FUNCTION_BLOCK FB_STI_Conveyor_V2 IMPLEMENTS ITF_SubsystemTransport
(**************************************************************************************
 * 	Application		:	BoxControl Framework
 *	Revision		:	$Revision: 355211 $
 *	Revision date	:	$Date: 2015-09-22 11:14:21 +0200 (Tue, 22 Sep 2015) $
 *	Last changed by	:	$Author: d7mangc $
 *	URL				:	$URL: http://almscdc.swisslog.com/repo/SWPD/Development/BoxControlFramework/20_Release/trunk/01_Software/BoxControlFramework/BoxControlFramework/JumpStart/11_Library/10_Application/11_Communication/12_MFCS/11_SIS/10_Base/FB_SIS_BaseDriver.TcPOU $
 *
 *	Purpose			:	Subsystem transport interface: Conveyor
 *
 * ------------------------------------------------------------------------------------
 *	Copyright Swisslog [IP AG], Switzerland. All rights reserved.
 * 
 * ------------------------------------------------------------------------------------
 *	
 * 	Revision History: 
 *
 * VERSION DATE         INITIALS     DESCRIPTION
 * 0.0     DD.MM.YYYY   (name)       (explain customized modifications)
 *
 **************************************************************************************)
VAR_INPUT
	Config					: ST_CFG_STI_Conveyor; // Config
END_VAR
VAR_OUTPUT
	Outputs					: ST_InOutputsSTI_Conveyor; // Outputs
END_VAR
VAR
	Init					: BOOL; // Initialize
	fbDebugMsg				: FB_DebugMsg; // Debug instance
	DebugMsg				: T_MAXSTRING; // Debug msg
	fbTCP_Driver			: FB_TCP_Driver;
	ErrorData				: ST_ErrorDataSet; // Error data
	DestinationPosition		: ST_PositionIdent; 
	Position				: ST_PositionIdent; 
	ExternalTU_DataIndex	: DINT; 
	TU_DataIndex			: DINT;
	TU_DataIndexAssignment	: DINT;
	LastHandoverTU_DataIndex: DINT;
	TransportControlData	: ST_TransportControlData; 
	eHandOverState			: E_HandoverState; // Handover state machine
	eLastHandOverState		: E_HandoverState; // Handover state machine
	eTakeOverState			: E_TakeoverState; // Takeover state machine
	eLastTakeOverState		: E_TakeoverState; // Takeover state machine
	Inputs					: ST_InOutputsSTI_Conveyor; // Input structure
	AdjTransportData		: ST_TransportData; // Transport data of adjacent function
	RecvByte				: ARRAY[1..38] OF BYTE; // Receive as bytes (alignment)
	SendByte				: ARRAY[1..38] OF BYTE; // Send as bytes (alignment)
	RecvData				: ST_STI_ConveyorData; // Incoming conveyor data
	SendData				: ST_STI_ConveyorData; // Outgoing conveyor data
	LastSendData			: ST_STI_ConveyorData; // Last outgoing conveyor data
	ReceivedDataLen			: UDINT; // Received length
	RecvCounter				: USINT; // Counts received messages
	SendCounter				: USINT; // Counts sent messages
	fbWatchdogTimer			: TON; // Monitors watchdog signal
	fbReinitConnection		: TON; // Timer connection retry
	fbResend				: TON; // Timer for resending last message
	fbHeartBeatTimer		: TON; // Timer for generating heart beat of watchdog
	TransportData			: ST_TransportData; // Transport data
	DataError				: BOOL; // Error on data allocation action
	FlagWatchdog			: BOOL; // Flag, to save last watchdog state
	tHeartBeat				: TIME; // Time for generating watchdog heart beat
	TU_ID_Present			: BOOL; // TU ID present
	AssignmentID_Present	: BOOL; // Assignment ID present
	NewIndexCreated			: BOOL;
	TTC						: ST_ITC_TTC; // TTC
END_VAR
VAR PERSISTENT
	Settings				: ST_CFG_STI_Conveyor;
END_VAR

(**************************************************************************************************************
   Body never called!
***************************************************************************************************************)
;

ACTION A_AllocateDataIndex:
(**************************************************************************************
 * 	NAME		A_AllocateDataIndex
 * 	FUNCTION	Allocate a data index
 **************************************************************************************)

 (**************************************************************************************
   Delete old
***************************************************************************************)
 // If an old index is still available
 IF ExternalTU_DataIndex <> 0 THEN
	// Check if a position contains this index
	Position := F_SearchPositionOfTU_Index(
					TU_DataIndex := ExternalTU_DataIndex,
					eStartFunctionNumber := E_FunctionNumber.F_BEGIN_FUNCTION);
					
	// If index was found on a position
	IF Position.eFunctionNumber > E_FunctionNumber.F_BEGIN_FUNCTION THEN
		// debug message: '11-001-0000-00-0,  used TU_DataIndex deleted, position = 99-999-9999-99-9,  TU_DataIndex = 5,  TuID = 000012345,  AssignmentID = 999999999'
		DebugMsg := '';
		DebugMsg := CONCAT(DebugMsg, F_AddDividerToSisString(SubsystemRegistry.SubsystemName));
		DebugMsg := CONCAT(DebugMsg, ',  used TU_DataIndex deleted');
		DebugMsg := CONCAT(DebugMsg, DebugTextBlocks.POSITION);
		DebugMsg := CONCAT(DebugMsg, Position.PositionName);
		DebugMsg := CONCAT(DebugMsg, F_CreateTU_DataString(TU_DataIndex:= ExternalTU_DataIndex));
		fbDebugMsg.M_SendWarningMsg(mMessage := DebugMsg);
		
		// Clear only index
		ExternalTU_DataIndex := 0;
	ELSE
		// debug message: '11-000-0000-00-0,  unused TU_DataIndex deleted, external = 99-999-9999-99-9,  TU_DataIndex = 5,  TuID = 000012345,  AssignmentID = 999999999'
		DebugMsg := '';
		DebugMsg := CONCAT(DebugMsg, F_AddDividerToSisString(SubsystemRegistry.SubsystemName));
		DebugMsg := CONCAT(DebugMsg, ',  unused TU_DataIndex deleted');
		DebugMsg := CONCAT(DebugMsg, DebugTextBlocks.POSITION);
		DebugMsg := CONCAT(DebugMsg, TO_STRING(Settings.eExternalFunctionNumber));  // ###todo: how to retrieve sis number string for external?
		DebugMsg := CONCAT(DebugMsg, F_CreateTU_DataString(TU_DataIndex:= ExternalTU_DataIndex));
		fbDebugMsg.M_SendInfoMsg(DebugMsg);
		// Clear data set
		F_DeleteTU_Data(
			TU_DataIndex 	:= ExternalTU_DataIndex,
			NoTTC 			:= TRUE);
			
		// Clear index
		ExternalTU_DataIndex := 0;
	END_IF
 END_IF
 
 (**************************************************************************************
   Allocate new index
***************************************************************************************)
TU_ID_Present := Inputs.TU_ID <> '000000000000000000' AND
				 Inputs.TU_ID <> '                  ' AND
			 	 Inputs.TU_ID <> '';

AssignmentID_Present := Inputs.AssignmentID > 0;

// If giving conveyor provides a TU ID or an assignment ID
IF TU_ID_Present OR
   AssignmentID_Present THEN
   
   // Reset
   DataError := FALSE;
   
	// Search if index based on TU-ID is already available 
	TU_DataIndex := F_SearchTU_ByHashCode(TU_ID := Inputs.TU_ID);
	// Search if index based on Assignment is already available
	TU_DataIndexAssignment := F_SearchAssignmentId(Inputs.AssignmentID);

	// When both an index for the TU-ID AND the Assignment ID is available in the system 
	IF TU_DataIndex > 0 AND TU_DataIndexAssignment > 0 THEN
		// Check if they are equal, otherwise data set is ignored
		// This would lead to a data mismatch.
		IF TU_DataIndex <> TU_DataIndexAssignment THEN
		   DataError := TRUE;
		   
		   	// Debug - wrong index found
			DebugMsg := CONCAT('External interface: AssignmentID and TU-ID have not the same index. TU-ID index:', DINT_TO_STRING(TU_DataIndex));
			DebugMsg := CONCAT(DebugMsg, ', AssignmentID index: ');
			DebugMsg := CONCAT(DebugMsg, DINT_TO_STRING(TU_DataIndexAssignment));
			fbDebugMsg.M_SendWarningMsg(mMessage := DebugMsg);
		
		// Clear TU slot before taking over TU data from the Interface
		ELSIF Settings.DeleteTU_Data THEN
			MEMSET(ADR(TU_DataTable[TU_DataIndex]), 0, SIZEOF(TU_DataTable[TU_DataIndex]));	
		END_IF 
		
	// When index for TU-ID OR  Assignment ID is available in the system
	ELSIF TU_DataIndex > 0  OR TU_DataIndexAssignment > 0 THEN
		
		IF Settings.DeleteTU_Data THEN
			// Clear TU slot before taking over TU data from the Interface
			MEMSET(ADR(TU_DataTable[TU_DataIndex]), 0, SIZEOF(TU_DataTable[TU_DataIndex]));	
		END_IF 
		
	// When index for Assignment ID is available in the system
	ELSIF TU_DataIndexAssignment > 0 THEN
		IF Settings.DeleteTU_Data THEN
			// Clear TU slot before taking over TU data from the Interface
			MEMSET(ADR(TU_DataTable[TU_DataIndexAssignment]), 0, SIZEOF(TU_DataTable[TU_DataIndexAssignment]));	
		END_IF 	
		TU_DataIndex := TU_DataIndexAssignment; 	
		
	ELSE
		// Allocate new one
	   TU_DataIndex := F_InsertTU_Data(
							eFunctionNumber := Settings.AdjFunctionNumber.eFunctionNumber,
							ZoneNumber := Settings.AdjFunctionNumber.ZoneNumber);
		
		NewIndexCreated := TU_DataIndex > 0;		
		
		// If creation was not succesfull
		IF NOT NewIndexCreated THEN
			DataError := TRUE;
		   
		   	// Debug - Image creation failed
			DebugMsg := 'External interface: AllocateDataIndex was not able to create free index';
			fbDebugMsg.M_SendWarningMsg(mMessage := DebugMsg);
			
			// Error no free TU Index
			IF ErrorData.ErrorType = E_ErrorType.NO_ERROR_PENDING THEN
				// Set communication error
				F_SetError(
					ErrorMsg	:= E_ErrorConv.NO_FREE_TU_DATA_SET,
					ErrorType 	:= E_ErrorType.ERROR,
					ErrorParam 	:= '',
					ErrorData	:= ErrorData);
			END_IF
		END_IF
	END_IF
   
	// When no error occured 
	IF NOT DataError AND 
		TU_DataIndex > 0 THEN
		
		//  when new Tu data index was created or exisitng should be overwritten
		IF	Settings.OverwriteTU_Data OR NewIndexCreated THEN
			//Takeover data from interface
			
			// Set data present
			TU_DataTable[TU_DataIndex].DataSet.DataPresent := TRUE;
			
			// Update data
			IF TU_ID_Present THEN
				TU_DataTable[TU_DataIndex].TU_ID.ASCII := Inputs.TU_ID;
				TU_DataTable[TU_DataIndex].TU_ID.HashCode := F_CreateHashCode(Inputs.TU_ID);
			END_IF
			
			IF AssignmentID_Present THEN
				TU_DataTable[TU_DataIndex].AssignmentID := Inputs.AssignmentID;
			END_IF
	
			IF Inputs.Destination <> '' THEN
				// Search function number of corresponding string
				DestinationPosition := F_SearchFunctionPosition(Position := Inputs.Destination);
			
				// Destination was found 
				IF DestinationPosition.eFunctionNumber <> 0 THEN
					TU_DataTable[TU_DataIndex].Destination[1].eFunctionNumber 	:= DestinationPosition.eFunctionNumber;
					TU_DataTable[TU_DataIndex].Destination[1].ZoneNumber 		:= DestinationPosition.ZoneNumber;
					TU_DataTable[TU_DataIndex].Destination[1].PositionName 		:= DestinationPosition.PositionName;
					TU_DataTable[TU_DataIndex].DataSet.JobPresent := TRUE;
					TU_DataTable[TU_DataIndex].DataSet.NumberOfDest := 1;
				ELSE
					// Debug - Destination not found
					DebugMsg := CONCAT('External interface: Destination not found(', Inputs.Destination);
					DebugMsg := CONCAT(DebugMsg, ')');
					
					fbDebugMsg.M_SendWarningMsg(mMessage := DebugMsg);
				END_IF
			END_IF			
		END_IF
		// Set to external TU Data Index
		ExternalTU_DataIndex := TU_DataIndex;
	END_IF
END_IF
END_ACTION

ACTION A_HandOverStates:
(**************************************************************************************
 * 	NAME		A_HandOverInterface
 * 	FUNCTION	Handover interface
 **************************************************************************************)

(**************************************************************************************
	Update outputs for external conveyor position
**************************************************************************************)
Outputs.ReadyToTakeOver := AdjTransportData.rTransportControlData.eTakeOverState = E_TakeOverState.READY OR
						   AdjTransportData.rTransportControlData.eTakeOverState = E_TakeOverState.INTERRUPTED;

Outputs.TakeoverStarted := AdjTransportData.rTransportControlData.eTakeOverState = E_TakeOverState.ACTIVE OR
						   AdjTransportData.rTransportControlData.eTakeOverState = E_TakeOverState.INTERRUPTED OR
						   AdjTransportData.rTransportControlData.eTakeOverState = E_TakeOverState.STOP OR
						   AdjTransportData.rTransportControlData.eTakeOverState = E_TakeOverState.COMPLETE;

Outputs.TakeoverActive := AdjTransportData.rTransportControlData.eTakeOverState = E_TakeOverState.ACTIVE;
						  
Outputs.TakeoverComplete := AdjTransportData.rTransportControlData.eTakeOverState = E_TakeOverState.COMPLETE;

Outputs.TransportActive := AdjTransportData.rTransportControlData.TransportActive;
Outputs.FastSpeedActive := AdjTransportData.rTransportControlData.FastSpeedActive;

(**************************************************************************************
	Simulates hand over state for external conveyor position
 **************************************************************************************)
CASE eHandOverState OF
	
	(**********************************************************************************
	   BEGIN
	***********************************************************************************)
	E_HandOverState.UNDEFINED:
	
		// Change state to "IDLE"
		eLastHandOverState := eHandOverState;
		eHandOverState := E_HandOverState.IDLE;
	
	(**********************************************************************************
	   IDLE
	***********************************************************************************)
	E_HandOverState.IDLE:

		// If external interface is ready to hand over
		IF Inputs.ReadyToHandOver THEN
			// Allocate data index
			A_AllocateDataIndex();
		
			// Change state to "IDLE"
			eLastHandOverState := eHandOverState;
			eHandOverState := E_HandOverState.READY;
		END_IF
	
	(**********************************************************************************
	   READY
	***********************************************************************************)
	E_HandOverState.READY:
	
		IF Inputs.HandoverActive THEN
			// Change state to "ACTIVE"
			eLastHandOverState := eHandOverState;
			eHandOverState := E_HandOverState.ACTIVE;
	
		// If external interface is not ready for hand over
		ELSIF NOT Inputs.ReadyToHandOver THEN
			// Go back to state to "IDLE"
			eLastHandOverState := eHandOverState;
			eHandOverState := E_HandOverState.IDLE;
		END_IF
		
	(**********************************************************************************
	   ACTIVE
	***********************************************************************************)
	E_HandOverState.ACTIVE:
	
		// Wait until completed
		IF Inputs.HandoverComplete THEN
			// Change state to "COMPLETE"
			eLastHandOverState := eHandOverState;
			eHandOverState := E_HandOverState.COMPLETE;
		
		// If handover is not active anymore
		ELSIF NOT Inputs.HandoverActive THEN
			// Ready already set -> Takeover conveyor stopped handover
			IF Inputs.ReadyToHandover THEN
				// Change state to "Interrupted"
				eLastHandOverState := eHandOverState;
				eHandOverState := E_HandOverState.INTERRUPTED;
				
			// Otherwise the external conveyor has stopped the handover
			ELSE
				// If the handover task is the same - was an error during transport -> Stop
				IF Inputs.HandoverStarted THEN
					// Change state to "Stop"
					eLastHandOverState := eHandOverState;
					eHandOverState := E_HandOverState.STOP;
					
				// Otherwise transport was aborted completely
				ELSE
					// Change state to "Idle"
					eLastHandOverState := eHandOverState;
					eHandOverState := E_HandOverState.IDLE;
				END_IF
			END_IF
		END_IF
	
	(**********************************************************************************
	   STOP
	***********************************************************************************)
	E_HandOverState.STOP:
			
		// Wait until transfer goes on 
		IF Inputs.HandoverActive THEN
			// Change state to "ACTIVE"
			eLastHandOverState := eHandOverState;
			eHandOverState := E_HandOverState.ACTIVE;

		// If the handover is completed 
		ELSIF Inputs.HandoverComplete THEN
			// Change state to "ACTIVE"
			eLastHandOverState := eHandOverState;
			eHandOverState := E_HandOverState.COMPLETE;	
		
		// If the ongoing transport task was aborted
		ELSIF NOT Inputs.HandoverStarted THEN
			// Change state to "Idle"
			eLastHandOverState := eHandOverState;
			eHandOverState := E_HandOverState.IDLE;
		END_IF
	
	(**********************************************************************************
	   INTERRUPTED
	***********************************************************************************)
	E_HandOverState.INTERRUPTED:
	
		// Wait until hadover is active
		IF Inputs.HandoverActive THEN
			// Change state to "ACTIVE"
			eLastHandOverState := eHandOverState;
			eHandOverState := E_HandOverState.ACTIVE;
			
		// If the handover is completed 
		ELSIF Inputs.HandoverComplete THEN
			// Change state to "ACTIVE"
			eLastHandOverState := eHandOverState;
			eHandOverState := E_HandOverState.COMPLETE;				
			
		// If the ongoing transport task was aborted
		ELSIF NOT Inputs.HandoverStarted THEN
			// Change state to "Idle"
			eLastHandOverState := eHandOverState;
			eHandOverState := E_HandOverState.IDLE;
		END_IF
		
	(**********************************************************************************
	   COMPLETE
	***********************************************************************************)
	E_HandOverState.COMPLETE:
	
		// Wait until transfer complete signal is resetted
		IF NOT Inputs.HandoverComplete OR
           NOT Inputs.HandoverStarted THEN
			// Change state to "IDLE"
			eLastHandOverState := eHandOverState;
			eHandOverState := E_HandOverState.IDLE;
		END_IF 
		
ELSE
	// Programming error
	DebugMsg := CONCAT(	'Programming error - Invalid state of external interface (Handover): ', 
					   	INT_TO_STRING(eHandOverState));
	DebugMsg := CONCAT(	DebugMsg, ' External connection : ');
	DebugMsg := CONCAT(	DebugMsg, INT_TO_STRING(Settings.eExternalFunctionNumber));
	fbDebugMsg.M_SendErrorMsg(DebugMsg);
END_CASE
END_ACTION

ACTION A_InputMapping:
(**************************************************************************************
 * 	NAME		A_InputMapping
 * 	FUNCTION	Map input variables
 **************************************************************************************)

(**************************************************************************************
   Map interface inputs
***************************************************************************************)
 
// If interface is configured as inbound
IF Settings.Inbound THEN
	Inputs.HandoverActive := RecvData.HandoverActive;
	Inputs.HandoverComplete := RecvData.HandoverComplete;
	Inputs.ReadyToHandover := RecvData.ReadyToHandover;	
	Inputs.HandoverStarted := RecvData.HandoverStarted;
	Inputs.TakeoverActive := FALSE;
	Inputs.TakeoverComplete := FALSE;
	Inputs.ReadyToTakeover := FALSE;
	Inputs.TakeoverStarted := FALSE;
	
// Otherwise, outbound
ELSE
	Inputs.TakeoverActive := RecvData.TakeoverActive;
	Inputs.TakeoverComplete := RecvData.TakeoverComplete;
	Inputs.ReadyToTakeover := RecvData.ReadyToTakeover;
	Inputs.TakeoverStarted := RecvData.TakeoverStarted;
	Inputs.HandoverActive := FALSE;
	Inputs.HandoverComplete := FALSE;
	Inputs.ReadyToHandover := FALSE;	
	Inputs.HandoverStarted := FALSE;
END_IF

// General data
Inputs.TU_ID := RecvData.TU_Data.TU_ID;
Inputs.AssignmentID := RecvData.TU_Data.AssignmentID;
Inputs.Destination := RecvData.TU_Data.Destination;

IF Settings.OnlyFastSpeed THEN
	Inputs.FastSpeedActive := TRUE;
ELSE
	Inputs.FastSpeedActive := RecvData.FastSpeedActive;
END_IF

Inputs.TransportActive := RecvData.TransportActive;

(**************************************************************************************
   Get external data
***************************************************************************************)
// Get transport data of adjacent function
AdjTransportData := F_GetAdjacentTransportData(
						eFunctionNumber 		:= Settings.AdjFunctionNumber.eFunctionNumber,
						eSourceFunctionNumber 	:= Settings.eExternalFunctionNumber);
END_ACTION

ACTION A_MonitorCommunication:
(**************************************************************************************
 * 	NAME		A_MonitorCommunication
 * 	FUNCTION	Monitors TCP Communication
 **************************************************************************************)

(**************************************************************************************
   Watchdog
***************************************************************************************) 
fbWatchdogTimer(IN := TRUE, PT := Settings.tWatchdog);
 
// If connection is server
IF Settings.TCP_Driver.Server THEN
	// Watchdog signals
	IF RecvData.WatchdogToggle = SendData.WatchdogToggle THEN
		// Reset timer
		fbWatchdogTimer(IN := FALSE);
		fbHeartBeatTimer(IN := TRUE, PT := tHeartBeat);
	END_IF
	
	fbHeartBeatTimer();
	IF fbHeartBeatTimer.Q THEN
		fbHeartBeatTimer(IN := FALSE);
		// Return watchdog signal
		SendData.WatchdogToggle := NOT RecvData.WatchdogToggle;
	END_IF

// Otherwise, client
ELSE
	// Watchdog signals
	IF RecvData.WatchdogToggle XOR SendData.WatchdogToggle THEN
		// Reset timer
		fbWatchdogTimer(IN := FALSE);
	END_IF
 	// Return watchdog signal
 	SendData.WatchdogToggle := RecvData.WatchdogToggle;
END_IF

(**************************************************************************************
   Reestablish connection
***************************************************************************************)
IF Settings.tRetryConnection <> T#0S THEN
	// Reestablish connection after a certain time
	fbReinitConnection(IN := fbWatchdogTimer.Q AND fbTCP_Driver.Connected, PT := Settings.tRetryConnection);
	
	// Restart
	IF fbReinitConnection.Q THEN
		fbTCP_Driver.M_RestartCom();
		// Reset
		fbReinitConnection(IN := FALSE);
	END_IF
ELSE
	// Reset
	fbReinitConnection(IN := FALSE);
END_IF

(**************************************************************************************
   Communication error
***************************************************************************************)
// Communication timeout
IF fbWatchdogTimer.Q AND
 	ErrorData.ErrorType = E_ErrorType.NO_ERROR_PENDING THEN
	// Set communication error
	F_SetError(
		ErrorMsg	:= E_ErrorConv.CONNECTION_ERROR_TO_EXTERNAL_INTERFACE,
		ErrorType 	:= E_ErrorType.ERROR,
		ErrorParam 	:= '',
		ErrorData	:= ErrorData);

// Communication reestablished
ELSIF NOT fbWatchdogTimer.Q AND ErrorData.ErrorCode.Conv = E_ErrorConv.CONNECTION_ERROR_TO_EXTERNAL_INTERFACE THEN
	// Auto reset
	F_ResetError(
		Reset		:= TRUE,
		ErrorData 	:= ErrorData);
END_IF
END_ACTION

ACTION A_OutputMapping:
(**************************************************************************************
 * 	NAME		A_OutputMapping
 * 	FUNCTION	Map output variables
 **************************************************************************************)

// If interface is configured as inbound
IF Settings.Inbound THEN
	SendData.TakeoverActive := Outputs.TakeoverActive;
	SendData.TakeoverComplete := Outputs.TakeoverComplete;
	SendData.ReadyToTakeover := Outputs.ReadyToTakeover;
	SendData.TakeoverStarted := Outputs.TakeoverStarted;
	SendData.HandoverActive := FALSE;
	SendData.HandoverComplete := FALSE;
	SendData.ReadyToHandover := FALSE;
	SendData.HandoverStarted := FALSE;
	
// Otherwise, outbound
ELSE
	SendData.HandoverActive := Outputs.HandoverActive;
	SendData.HandoverStarted := Outputs.HandoverStarted;
	SendData.HandoverComplete := Outputs.HandoverComplete;
	SendData.ReadyToHandover := Outputs.ReadyToHandover;
	SendData.TakeoverActive := FALSE;
	SendData.TakeoverComplete := FALSE;
	SendData.ReadyToTakeover := FALSE;
	SendData.TakeoverStarted := FALSE;
END_IF

// General data
SendData.TU_Data.TU_ID := Outputs.TU_ID;
SendData.TU_Data.AssignmentID := Outputs.AssignmentID;
SendData.TU_Data.Destination := Outputs.Destination;
SendData.FastSpeedActive := Outputs.FastSpeedActive;
SendData.TransportActive := Outputs.TransportActive;
END_ACTION

ACTION A_TakeOverStates:
(**************************************************************************************
 * 	NAME		A_TakeOverInterface
 * 	FUNCTION	TakeOver interface - Take over from external conveyor
 **************************************************************************************)

 (**************************************************************************************
	Update outputs for external conveyor position
 **************************************************************************************)
Outputs.ReadyToHandover := AdjTransportData.rTransportControlData.eHandOverState = E_HandOverState.READY OR
						   AdjTransportData.rTransportControlData.eHandOverState = E_HandOverState.INTERRUPTED;

Outputs.HandoverStarted := AdjTransportData.rTransportControlData.eHandOverState = E_HandOverState.ACTIVE OR
						   AdjTransportData.rTransportControlData.eHandOverState = E_HandOverState.INTERRUPTED OR
						   AdjTransportData.rTransportControlData.eHandOverState = E_HandOverState.STOP OR
						   AdjTransportData.rTransportControlData.eHandOverState = E_HandOverState.COMPLETE;

Outputs.HandoverActive := AdjTransportData.rTransportControlData.eHandOverState = E_HandOverState.ACTIVE;
						  
Outputs.HandoverComplete := AdjTransportData.rTransportControlData.eHandOverState = E_HandOverState.COMPLETE;

TU_DataIndex := AdjTransportData.rTransportControlData.TU_DataIndex;
	
IF TU_DataIndex > 0 THEN				
	Outputs.Destination := TU_DataTable[TU_DataIndex].Destination[1].PositionName;
ELSE
	Outputs.Destination := '';
END_IF							

Outputs.TU_ID := TU_DataTable[TU_DataIndex].TU_ID.ASCII;
Outputs.AssignmentID := TU_DataTable[TU_DataIndex].AssignmentID;
Outputs.TransportActive := AdjTransportData.rTransportControlData.TransportActive;
Outputs.FastSpeedActive := AdjTransportData.rTransportControlData.FastSpeedActive;

(**************************************************************************************
	Simulates take over state from external conveyor position
 **************************************************************************************)
CASE eTakeOverState OF
	
	(**********************************************************************************
	   BEGIN
	***********************************************************************************)
	E_TakeOverState.UNDEFINED:
	
		// Change state to "IDLE"
		eLastTakeOverState := eTakeOverState;
		eTakeOverState := E_TakeOverState.IDLE;
	
	(**********************************************************************************
	   IDLE
	***********************************************************************************)
	E_TakeOverState.IDLE:
	
		// If external interface is ready to take over
		IF Inputs.ReadyToTakeover THEN
			// Change state to "READY"
			eLastTakeOverState := eTakeOverState;
			eTakeOverState := E_TakeOverState.READY;
		END_IF
		
	(**********************************************************************************
	   READY
	***********************************************************************************)
	E_TakeOverState.READY:

		IF Inputs.HandoverActive THEN
			// Change state to "ACTIVE"
			eLastHandOverState := eHandOverState;
			eHandOverState := E_HandOverState.ACTIVE;
	
		// If external interface is not ready for hand over
		ELSIF NOT Inputs.ReadyToHandOver THEN
			// Go back to state to "IDLE"
			eLastHandOverState := eHandOverState;
			eHandOverState := E_HandOverState.IDLE;
		END_IF
	
	(**********************************************************************************
	   ACTIVE
	***********************************************************************************)
	E_TakeOverState.ACTIVE:
	
		// Wait until completed
		IF Inputs.TakeoverComplete THEN
			// Change state to "COMPLETE"
			eLastTakeOverState := eTakeOverState;
			eTakeOverState := E_TakeOverState.COMPLETE;
			
		// If takeover is not active anymore
		ELSIF NOT Inputs.TakeoverActive THEN
			// Ready already set - Interupted as reason of other conveyor
			IF Inputs.ReadyToTakeover THEN
				// Change state to "interrupted"
				eLastTakeOverState := eTakeOverState;
				eTakeOverState := E_TakeOverState.INTERRUPTED;
			ELSE
				// If the takeover task is the same - was an error during transport -> Stop
				IF Inputs.TakeoverStarted THEN
					// Change state to "Stop"
					eLastTakeOverState := eTakeOverState;
					eTakeOverState := E_TakeOverState.STOP;
					
				// Otherwise transport was aborted completely
				ELSE
					// Change state to "Idle"
					eLastTakeOverState := eTakeOverState;
					eTakeOverState := E_TakeOverState.IDLE;
				END_IF
			END_IF
		END_IF
	
	(**********************************************************************************
	   STOP
	***********************************************************************************)
	E_TakeOverState.STOP:
	
		// Wait until transfer goes on
		IF Inputs.TakeoverActive THEN
			// Change state to "ACTIVE"
			eLastTakeOverState := eTakeOverState;
			eTakeOverState := E_TakeOverState.ACTIVE;

		// If the takeover is completed 
		ELSIF Inputs.TakeoverComplete THEN
			// Change state to "ACTIVE"
			eLastTakeOverState := eTakeOverState;
			eTakeOverState := E_TakeOverState.COMPLETE;				
			
		ELSIF NOT Inputs.TakeoverStarted THEN
			// Change state to "Idle"
			eLastTakeOverState := eTakeOverState;
			eTakeOverState := E_TakeOverState.IDLE;
		END_IF
	
	(**********************************************************************************
	   INTERRUPTED
	***********************************************************************************)
	E_TakeOverState.INTERRUPTED:
	
		// Wait until transfer goes on
		IF Inputs.TakeoverActive THEN
			// Change state to "ACTIVE"
			eLastTakeOverState := eTakeOverState;
			eTakeOverState := E_TakeOverState.ACTIVE;
		
		// If the takeover is completed 
		ELSIF Inputs.TakeoverComplete THEN
			// Change state to "ACTIVE"
			eLastTakeOverState := eTakeOverState;
			eTakeOverState := E_TakeOverState.COMPLETE;		
			
		ELSIF NOT Inputs.TakeoverStarted THEN
			// Change state to "Idle"
			eLastTakeOverState := eTakeOverState;
			eTakeOverState := E_TakeOverState.IDLE;
		END_IF
	
	(**********************************************************************************
	   COMPLETE
	***********************************************************************************)
	E_TakeOverState.COMPLETE:
	
		// Wait until transfer complete signal is resetted
		IF NOT Inputs.TakeoverComplete OR
           NOT Inputs.TakeoverStarted THEN
			// Change state to "IDLE"
			eLastTakeOverState := eTakeOverState;
			eTakeOverState := E_TakeOverState.IDLE;
		END_IF 
	
ELSE
	// Programming error
	DebugMsg := CONCAT(	'Programming error - Invalid state of external interface (Takeover): ', 
					   	INT_TO_STRING(eTakeOverState));
	DebugMsg := CONCAT(	DebugMsg, ' External connection : ');
	DebugMsg := CONCAT(	DebugMsg, INT_TO_STRING(Settings.eExternalFunctionNumber));
	fbDebugMsg.M_SendErrorMsg(DebugMsg);
END_CASE
END_ACTION

ACTION A_TCP_Communication:
(**************************************************************************************
 * 	NAME		A_TCP_Communication
 * 	FUNCTION	Handles TCP Communication to external interface
 **************************************************************************************)

 // Call driver
 fbTCP_Driver(
	Config 			:= Settings.TCP_Driver,
	pReceiveData 	:= ADR(RecvByte),
	ReceiveDataLen 	:= SIZEOF(RecvByte),
	ReceivedBytes	=> ReceivedDataLen);
 
(**************************************************************************************
   Receive data
***************************************************************************************)
// Check TCP/IP channel for new data
IF fbTCP_Driver.NewData THEN
	// Check border counter
	IF RecvCounter > 254 THEN
		// Reset
		RecvCounter := 0;
	END_IF
	
	// Update counter
	RecvCounter := RecvCounter + 1;
	
	// Fits the data length	
	IF ReceivedDataLen <> SIZEOF(RecvByte) THEN
		// Wrong value
		F_SetError(
			ErrorMsg	:= E_ErrorConv.WRONG_VALUE,
			ErrorType 	:= E_ErrorType.ERROR,
			ErrorParam 	:= '',
			ErrorData	:= ErrorData);
			
	ELSE
		// Map values - (alignment to ensure compatibility to other systems)
		RecvData.WatchdogToggle 	:= RecvByte[1].0;
		RecvData.ReadyToTakeover	:= RecvByte[1].1;
		RecvData.TakeoverStarted 	:= RecvByte[1].2;
		RecvData.TakeoverActive 	:= RecvByte[1].3;
		RecvData.TakeoverComplete 	:= RecvByte[1].4;
		RecvData.ReadyToHandover 	:= RecvByte[1].5;
		RecvData.HandoverStarted 	:= RecvByte[1].6;
		RecvData.HandoverActive 	:= RecvByte[1].7;
		
		RecvData.HandoverComplete 	:= RecvByte[2].0;
		RecvData.FastSpeedActive 	:= RecvByte[2].1;
		RecvData.TransportActive 	:= RecvByte[2].2;
		RecvData.Reserve1 			:= RecvByte[2].3;
		RecvData.Reserve2 			:= RecvByte[2].4;
		RecvData.Reserve3 			:= RecvByte[2].5;
		RecvData.Reserve4 			:= RecvByte[2].6;
		RecvData.Reserve5 			:= RecvByte[2].7;
		
		MEMCPY(destAddr := ADR(RecvData.TU_Data), srcAddr := ADR(RecvByte[3]), n := SIZEOF(RecvData.TU_Data));
	END_IF
	
	// Data processed
	fbTCP_Driver.M_DataProcessed();
END_IF

(**************************************************************************************
   Send data
***************************************************************************************)
// If the connection is established
IF fbTCP_Driver.Connected THEN
	// Call message resend timer
	fbResend(IN := Settings.tResendMsg <> T#0S, PT := Settings.tResendMsg);
	
	// If data have changed or resend is requested
	IF (MEMCMP(
		pBuf1 := ADR(LastSendData),
		pBuf2 := ADR(SendData),
		n	  := SIZEOF(SendData)) <> 0 OR fbResend.Q) AND NOT fbTCP_Driver.SendBusy THEN
	
		LastSendData := SendData;
		
		// Reset timer
		fbResend(IN := FALSE);
		
		// Map values - (alignment to ensure compatibility to other systems)
		SendByte[1].0 := SendData.WatchdogToggle;
		SendByte[1].1 := SendData.ReadyToTakeover;
		SendByte[1].2 := SendData.TakeoverStarted;
		SendByte[1].3 := SendData.TakeoverActive;
		SendByte[1].4 := SendData.TakeoverComplete;
		SendByte[1].5 := SendData.ReadyToHandover;
		SendByte[1].6 := SendData.HandoverStarted;
		SendByte[1].7 := SendData.HandoverActive;
		
		SendByte[2].0 := SendData.HandoverComplete;
		SendByte[2].1 := SendData.FastSpeedActive;
		SendByte[2].2 := SendData.TransportActive;
		SendByte[2].3 := SendData.Reserve1;
		SendByte[2].4 := SendData.Reserve2;
		SendByte[2].5 := SendData.Reserve3;
		SendByte[2].6 := SendData.Reserve4;
		SendByte[2].7 := SendData.Reserve5;
		
		MEMCPY(destAddr := ADR(SendByte[3]), srcAddr := ADR(SendData.TU_Data), n := SIZEOF(SendData.TU_Data));
		
		// Check border counter
		IF SendCounter > 254 THEN
			// Reset
			SendCounter := 0;
		END_IF
			
		// Update message counter
		SendCounter := SendCounter + 1;
	
		// Forward data to TCP channel
		fbTCP_Driver.M_Send(
			mpSendData := ADR(SendByte),
			mSendDataLen := SIZEOF(SendByte));
	END_IF
ELSE
	// Reset
	fbResend(IN := FALSE);
END_IF
END_ACTION

METHOD M_CallInterface : BOOL
(**************************************************************************************
 * 	Application		:	BoxControl Framework
 *	Revision		:	$Revision: 355136 $
 *	Revision date	:	$Date: 2015-09-21 07:38:56 +0200 (Mo, 21 Sep 2015) $
 *	Last changed by	:	$Author: d7mangc $
 *	URL				:	$URL: http://almscdc.swisslog.com/repo/SWPD/Development/BoxControlFramework/20_Release/trunk/01_Software/BoxControlFramework/BoxControlFramework/JumpStart/11_Library/10_Application/12_ElementFunctions/10_Functions/FB_TransportControl.TcPOU $
 *
 *	Purpose			:	Call main interface
 *
 * ------------------------------------------------------------------------------------
 *	Copyright Swisslog [IP AG], Switzerland. All rights reserved.
 * 
 * ------------------------------------------------------------------------------------
 *	
 * 	Revision History: 
 *
 * 	VERSION			DATE			INITIALS			DESCRIPTION
 *	0.1				01.01.2001		swl					Example
 *
 **************************************************************************************)
VAR_IN_OUT
	mErrorData				: ST_ErrorDataSet; // Error data
END_VAR

// Store inputs in instance
ErrorData := mErrorData;

(**************************************************************************************
	Init
 **************************************************************************************)
M_Init(mInit := FALSE);

(**************************************************************************************
	General error reset
 **************************************************************************************)
F_ResetError(
	Reset		:= FALSE,
	ErrorData 	:= ErrorData);

(***********************************************************************************
Monitor TCP/IP communication
***********************************************************************************)
A_MonitorCommunication();

(***********************************************************************************
TCP/IP communication
***********************************************************************************)
A_TCP_Communication();

(**************************************************************************************
	Input mapping
 **************************************************************************************)
A_InputMapping();

(**************************************************************************************
	Transport interface - Handles external conveyor position
 **************************************************************************************)
IF Settings.Inbound THEN
	// Incoming - Handle hand over states
	//			<---
	//  TakeOver  |	   HandOver
	// |-------|  |   |--------|
	//	 INTERN	  |		EXTERN
	A_HandOverStates();
	
ELSE
	// Outgoing - Handle take over states
	//			--->
	//  HandOver  |	   TakeOver
	// |-------|  |   |--------|
	//	 INTERN	  |		EXTERN
	A_TakeOverStates();
END_IF


(**************************************************************************************
	Output mapping
 **************************************************************************************)
A_OutputMapping();

// Update error structure
mErrorData := ErrorData;
END_METHOD

METHOD PROTECTED M_DoMoveTuDataIndex

VAR
	LastHandoverTU_DataIndex: DINT;
END_VAR
// External conveyor took index over - remove on giving position
LastHandoverTU_DataIndex := F_MoveTU_DataIndex(
								eFunctionNumber := Settings.AdjFunctionNumber.eFunctionNumber,
								mZoneNumber 	:= Settings.AdjFunctionNumber.ZoneNumber);
					
// If a index was found and outimage is active
IF LastHandoverTU_DataIndex <> 0 AND Settings.DeleteTU_Data THEN

	// Update "last known position"		
	TU_DataTable[LastHandoverTU_DataIndex].TimeStamp.eInsertFunctionNumber:=Settings.AdjFunctionNumber.eFunctionNumber;
	TU_DataTable[LastHandoverTU_DataIndex].TimeStamp.InsertZoneNumber:= Settings.AdjFunctionNumber.ZoneNumber;	

	// debug message
	// example: '11-002-1979-09-1,  TU leaving subsystem,  destination = 33-044-1979-01-9,  TU_DataIndex = 3,  TuID = 123456,  AssignmentID = 987654321'
	DebugMsg:= '';
	DebugMsg:= CONCAT(DebugMsg, F_AddDividerToSisString(Settings.AdjFunctionNumber.PositionName));
	DebugMsg:= CONCAT(DebugMsg, ',  TU leaving subsystem');
	DebugMsg:= CONCAT(DebugMsg, DebugTextBlocks.DESTINATION);
	DebugMsg:= CONCAT(DebugMsg, TO_STRING(Settings.eExternalFunctionNumber) );
	DebugMsg:= CONCAT(DebugMsg, F_CreateTU_DataString(TU_DataIndex:= LastHandoverTU_DataIndex) );
	fbDebugMsg.M_SendInfoMsg(mMessage := DebugMsg);

	// inform warehouse management (TTC) 
	IF NOT Settings.SuppressTTC THEN
		TTC.Position    := F_ReduceToAlphaNumeric(InputString := Settings.AdjFunctionNumber.PositionName); 					
		TTC.TU_DataIndex:= TU_DataIndex;
		TTC.MsgSequence := 0;
		TTC.TU_ID       := TU_DataTable[LastHandoverTU_DataIndex].TU_ID.ASCII;
		TTC.AssignmentID:= TU_DataTable[LastHandoverTU_DataIndex].AssignmentID;
		TTC.ReturnCode  := E_ErrorConv.TU_LEFT_SUBSYSTEM;
		System.fbITC_Manager.M_SendData(meChannel:= 0, 
										mMsgType := E_ITC_MsgTypeConv.TRANSPORT_TASK_COMPLETE, 
										mpData   := ADR(TTC),
										mLen     := SIZEOF(TTC));
	END_IF

	// Delete image in own system
	F_DeleteTU_Data(TU_DataIndex:= LastHandoverTU_DataIndex,
					NoTTC       := TRUE);
END_IF
END_METHOD

METHOD M_GetTransportData : REFERENCE TO ST_TransportData
(**************************************************************************************
 * 	Application		:	BoxControl Framework
 *	Revision		:	$Revision: 355211 $
 *	Revision date	:	$Date: 2015-09-22 11:14:21 +0200 (Tue, 22 Sep 2015) $
 *	Last changed by	:	$Author: d7mangc $
 *	URL				:	$URL: http://almscdc.swisslog.com/repo/SWPD/Development/BoxControlFramework/20_Release/trunk/01_Software/BoxControlFramework/BoxControlFramework/JumpStart/11_Library/10_Application/11_Communication/12_MFCS/11_SIS/10_Base/FB_SIS_BaseDriver.TcPOU $
 *
 *	Purpose			:	Return transport data
 *
 * ------------------------------------------------------------------------------------
 *	Copyright Swisslog [IP AG], Switzerland. All rights reserved.
 * 
 * ------------------------------------------------------------------------------------
 *	
 * 	Revision History: 
 *
 * 	VERSION			DATE			INITIALS			DESCRIPTION
 *	0.1				01.01.2001		swl					Example
 *
 **************************************************************************************)
// Prepare transport control data
TransportControlData.eHandOverState := eHandOverState;
TransportControlData.eTakeOverState := eTakeOverState;
TransportControlData.FastSpeedActive := Inputs.FastSpeedActive;
TransportControlData.TransportActive := Inputs.TransportActive;

// Return
TransportData.eFunctionNumber := Settings.eExternalFunctionNumber;
TransportData.ZoneNumber := 0;
MEMSET(ADR(TransportData.rSettings), 0, SIZEOF(TransportData.rSettings));
TransportData.rTransportControlData REF= TransportControlData;
M_GetTransportData REF= TransportData;
END_METHOD

METHOD M_Init : BOOL
(**************************************************************************************
 * 	Application		:	BoxControl Framework
 *	Revision		:	$Revision: 355211 $
 *	Revision date	:	$Date: 2015-09-22 11:14:21 +0200 (Tue, 22 Sep 2015) $
 *	Last changed by	:	$Author: b7bolm $
 *	URL				:	$URL: http://almscdc.swisslog.com/repo/SWPD/Development/BoxControlFramework/20_Release/trunk/01_Software/BoxControlFramework/BoxControlFramework/JumpStart/11_Library/10_Application/11_Communication/12_MFCS/11_SIS/10_Base/FB_SIS_BaseDriver.TcPOU $
 *
 *	Purpose			:	Initialize interface
 *
 * ------------------------------------------------------------------------------------
 *	Copyright Swisslog [IP AG], Switzerland. All rights reserved.
 * 
 * ------------------------------------------------------------------------------------
 *	
 * 	Revision History: 
 *
 * 	VERSION			DATE			INITIALS			DESCRIPTION
 *	0.1				01.01.2001		swl					Example
 *
 **************************************************************************************)
VAR_INPUT
	mInit			: BOOL; // Force init
END_VAR

IF NOT Init THEN
	
	Settings := Config;

	// Set default value if not configured
	IF Settings.tHeartBeat = T#0S THEN
		tHeartBeat := T#1S;
	ELSE
		tHeartBeat := Settings.tHeartBeat;
	END_IF

	Init := TRUE;
END_IF
END_METHOD

METHOD M_MoveTU_DataIndex : DINT
(**************************************************************************************
 * 	Application		:	BoxControl Framework
 *	Revision		:	$Revision: 355211 $
 *	Revision date	:	$Date: 2015-09-22 11:14:21 +0200 (Tue, 22 Sep 2015) $
 *	Last changed by	:	$Author: b7bolm $
 *	URL				:	$URL: http://almscdc.swisslog.com/repo/SWPD/Development/BoxControlFramework/20_Release/trunk/01_Software/BoxControlFramework/BoxControlFramework/JumpStart/11_Library/10_Application/11_Communication/12_MFCS/11_SIS/10_Base/FB_SIS_BaseDriver.TcPOU $
 *
 *	Purpose			:	Initialize interface
 *
 * ------------------------------------------------------------------------------------
 *	Copyright Swisslog [IP AG], Switzerland. All rights reserved.
 * 
 * ------------------------------------------------------------------------------------
 *	
 * 	Revision History: 
 *
 * 	VERSION			DATE			INITIALS			DESCRIPTION
 *	0.1				01.01.2001		swl					Example
 *
 **************************************************************************************)
// Return TU Data Index
M_MoveTU_DataIndex := ExternalTU_DataIndex;

// Clear internally
ExternalTU_DataIndex := 0;
END_METHOD

END_FUNCTION_BLOCK

(* stored: Version 1.1.0.1, ProductVersion 3.1.4024.4
   POU FB_STI_Conveyor_V2: Id {7c1e2f3d-6362-4fa3-82af-ae892eb2f034}, SpecialFunc None
   Action A_AllocateDataIndex: Id {bafd0bb4-4999-4767-a6f8-7cfdb6733b64}
   Action A_HandOverStates: Id {9601d5b6-6d1f-4ed0-9e09-0a9da6d88600}
   Action A_InputMapping: Id {47772434-9f98-44e1-8d47-0b8f80acd83f}
   Action A_MonitorCommunication: Id {f97ed628-7803-4445-9142-94eee5be8480}
   Action A_OutputMapping: Id {1031f6ab-7ba0-4d6b-a2be-527f93a34eed}
   Action A_TakeOverStates: Id {2cd9e415-05d3-47b7-8617-e5017642c2e0}
   Action A_TCP_Communication: Id {fa80b70e-7826-4ffd-8448-5908a6ea3a8c}
   Method M_CallInterface: Id {492a1533-3323-497b-98f2-a9339ae34934}
   Method M_DoMoveTuDataIndex: Id {30459d82-abb2-4f58-b426-3e5d79b1e05e}
   Method M_GetTransportData: Id {690e9779-2657-463b-966c-ee836936a9aa}
   Method M_Init: Id {8b34a706-804f-4287-bff2-8e7ad140e929}
   Method M_MoveTU_DataIndex: Id {cd1bbf7c-dbe4-4ea0-b34e-04a1ab44a380} *)
